KUKA KRL program: nplacestr16RS2.src, nplacestr16RS2.dat

--- nplacestr16RS2.src ---
&ACCESS RVP
&REL 1
&PARAM TEMPLATE = C:\KRC\Roboter\Template\ExpertVorgabe
&PARAM EDITMASK = *
DEF nplacestr16RS2( )
;FOLD INI
  ;FOLD BASISTECH INI
    GLOBAL INTERRUPT DECL 3 WHEN $STOPMESS==TRUE DO IR_STOPM ( )
    INTERRUPT ON 3
    BAS (#INITMOV,0 )
  ;ENDFOLD (BASISTECH INI)
  ;FOLD USER INI
    ;Make your modifications here

  ;ENDFOLD (USER INI)
;ENDFOLD (INI)




SWITCH NumCuring

;*******************************************************
CASE 91601
;*******************************************************
;*** Utilizar para hacer touchup en ptp a continuacion ***;
; 1  Ejecutar Axis_Rob_Move
; 2  Hacer TouchUp en ptp
; 3  Eliminar Axis_Rob_Move y comentarios

Axis_Rob_Move(1.69,-82.8,66.93,14.32,12.14,193,70,50)

;FOLD PTP pWB91601RS2 Vel=100 % PDAT_MESA Tool[10]:AMF1_G1000 Base[7]:BWB4S2;%{PE}%R 5.5.32,%MKUKATPBASIS,%CMOVE,%VPTP,%P 1:PTP, 2:pWB91601RS2, 3:, 5:100, 7:PDAT_MESA
$BWDSTART=FALSE
PDAT_ACT=PPDAT_MESA
FDAT_ACT=FpWB91601RS2
BAS(#PTP_PARAMS,100)
PTP XpWB91601RS2
;ENDFOLD
;*********************************************************;

;***Axis_Rob_Move de ayuda para aproximarse a dejada ***;
; Borrar tras touchup en LIN de dejada
Axis_Rob_Move(-90.22,-57.13,49.23,-5.44,97.37,193.9,20,50)
;*******************************************************;

PTP_OFFS(XP91601RS2, FP91601RS2, 0, -450, 30, 0, 0, 0, #TOOL, 20, 50, 0.0)

Cicle_Grp_M1000 (Inic_Pla_Right)

;***borrar***;
cyltopos(prg_200)
halt
;************;

LIN_OFFS(XP91601RS2, FP91601RS2, 0, 0, 30, 0, 0, 0, #TOOL, 0.1, 50, 0.0)
LIN_OFFS(XP91601RS2, FP91601RS2, 0, 0, 15, 0, 0, 0, #TOOL, 0.1, 50, 0.0)

Cntr_Grp_M1000 (C05C06,RH)

;FOLD LIN P91601RS2 Vel=0.1 m/s LV020Z0 Tool[10]:AMF1_G1000 Base[7]:BWB4S2;%{PE}%R 5.5.32,%MKUKATPBASIS,%CMOVE,%VLIN,%P 1:LIN, 2:P91601RS2, 3:, 5:0.1, 7:V020Z0
$BWDSTART=FALSE
LDAT_ACT=LV020Z0
FDAT_ACT=FP91601RS2
BAS(#CP_PARAMS,0.1)
LIN XP91601RS2
;ENDFOLD

Cntr_Grp_M1000 (AMF09,RLS)
Cyltopos (PRG_51)
Cntr_Grp_M1000 (C07C08,RH)
Cyltopos (PRG_61)
Cntr_Grp_M1000 (AMF10,RLS)
Cntr_Grp_M1000 (C05C06,FREE)
Cntr_Grp_M1000 (C07C08,FREE)
Cyltopos(PRG_88)
LIN_REL{Z -20}#TOOL
Cyltopos (PRG_105)
LIN_REL{Z -30}#TOOL
Cyltopos (PRG_200)

;*** MOVIMIENTOS DE OFFSETS ***;

LIN_OFFS(XP91601RS2, FP91601RS2, 0, 0, -50, 0, 0, 0, #TOOL, 0.3, 50, 0.0)
LIN_OFFS(XP91601RS2, FP91601RS2, 0, -450, -50, 0, 0, 0, #TOOL, 0.3, 50, 0.0)


;******* MEDICION LASER *******;

LIN_OFFS(XPLAS91601RS2_1, FPLAS91601RS2_1, 0, -200, 0, 0, 0, 0, #TOOL, 0.3, 50, 0.0)

cyltopos (prg_61)

;FOLD LIN PLAS91601RS2_1 Vel=0.3 m/s LV020Z0 Tool[10]:AMF1_G1000 Base[7]:BWB4S2;%{PE}%R 5.5.32,%MKUKATPBASIS,%CMOVE,%VLIN,%P 1:LIN, 2:PLAS91601RS2_1, 3:, 5:0.3, 7:V020Z0
$BWDSTART=FALSE
LDAT_ACT=LV020Z0
FDAT_ACT=FPLAS91601RS2_1
BAS(#CP_PARAMS,0.3)
LIN XPLAS91601RS2_1
;ENDFOLD

;Movimimiento de busqueda con laser
;Search( , )

;FOLD LIN PLAS91601RS2_2 Vel=0.3 m/s LV020Z0 Tool[10]:AMF1_G1000 Base[7]:BWB4S2;%{PE}%R 5.5.32,%MKUKATPBASIS,%CMOVE,%VLIN,%P 1:LIN, 2:PLAS91601RS2_2, 3:, 5:0.3, 7:V020Z0
$BWDSTART=FALSE
LDAT_ACT=LV020Z0
FDAT_ACT=FPLAS91601RS2_2
BAS(#CP_PARAMS,0.3)
LIN XPLAS91601RS2_2
;ENDFOLD


;Movimimiento de busqueda con laser
;Search( , )

LIN_OFFS(XPLAS91601RS2_1, FPLAS91601RS2_1, 0, -200, 0, 0, 0, 0, #TOOL, 0.3, 50, 0.0)

;******************************;

;FOLD PTP pWB91601RS2 Vel=100 % PDAT_MESA Tool[10]:AMF1_G1000 Base[7]:BWB4S2;%{PE}%R 5.5.32,%MKUKATPBASIS,%CMOVE,%VPTP,%P 1:PTP, 2:pWB91601RS2, 3:, 5:100, 7:PDAT_MESA
$BWDSTART=FALSE
PDAT_ACT=PPDAT_MESA
FDAT_ACT=FpWB91601RS2
BAS(#PTP_PARAMS,100)
PTP XpWB91601RS2
;ENDFOLD

;*******************************************************
CASE 91603
;*******************************************************
;*** Utilizar para hacer touchup en ptp a continuacion ***;
; 1  Ejecutar Axis_Rob_Move
; 2  Hacer TouchUp en ptp
; 3  Eliminar Axis_Rob_Move y comentarios

Axis_Rob_Move(1.69,-82.8,66.93,14.32,12.14,193,70,50)

;FOLD PTP pWB91603RS2 Vel=100 % PDAT_MESA Tool[10]:AMF1_G1000 Base[7]:BWB4S2;%{PE}%R 5.5.32,%MKUKATPBASIS,%CMOVE,%VPTP,%P 1:PTP, 2:pWB91603RS2, 3:, 5:100, 7:PDAT_MESA
$BWDSTART=FALSE
PDAT_ACT=PPDAT_MESA
FDAT_ACT=FpWB91603RS2
BAS(#PTP_PARAMS,100)
PTP XpWB91603RS2
;ENDFOLD
;*********************************************************;

;***Axis_Rob_Move de ayuda para aproximarse a dejada ***;
; Borrar tras touchup en LIN de dejada
Axis_Rob_Move(-90.22,-57.13,49.23,-5.44,97.37,193.9,20,50)
;*******************************************************;

PTP_OFFS(XP91603RS2, FP91603RS2, 0, -450, 30, 0, 0, 0, #TOOL, 20, 50, 0.0)

Cicle_Grp_M1000 (Inic_Pla_Right)

;***borrar***;
cyltopos(prg_200)
halt
;************;

LIN_OFFS(XP91603RS2, FP91603RS2, 0, 0, 30, 0, 0, 0, #TOOL, 0.1, 50, 0.0)
LIN_OFFS(XP91603RS2, FP91603RS2, 0, 0, 15, 0, 0, 0, #TOOL, 0.1, 50, 0.0)

Cntr_Grp_M1000 (C05C06,RH)

;FOLD LIN P91603RS2 Vel=0.1 m/s LV020Z0 Tool[10]:AMF1_G1000 Base[7]:BWB4S2;%{PE}%R 5.5.32,%MKUKATPBASIS,%CMOVE,%VLIN,%P 1:LIN, 2:P91603RS2, 3:, 5:0.1, 7:V020Z0
$BWDSTART=FALSE
LDAT_ACT=LV020Z0
FDAT_ACT=FP91603RS2
BAS(#CP_PARAMS,0.1)
LIN XP91603RS2
;ENDFOLD

Cntr_Grp_M1000 (AMF09,RLS)
Cyltopos (PRG_51)
Cntr_Grp_M1000 (C07C08,RH)
Cyltopos (PRG_61)
Cntr_Grp_M1000 (AMF10,RLS)
Cntr_Grp_M1000 (C05C06,FREE)
Cntr_Grp_M1000 (C07C08,FREE)
Cyltopos(PRG_88)
LIN_REL{Z -20}#TOOL
Cyltopos (PRG_105)
LIN_REL{Z -30}#TOOL
Cyltopos (PRG_200)

;*** MOVIMIENTOS DE OFFSETS ***;

LIN_OFFS(XP91603RS2, FP91603RS2, 0, 0, -50, 0, 0, 0, #TOOL, 0.3, 50, 0.0)
LIN_OFFS(XP91603RS2, FP91603RS2, 0, -450, -50, 0, 0, 0, #TOOL, 0.3, 50, 0.0)


;******* MEDICION LASER *******;

LIN_OFFS(XPLAS91603RS2_1, FPLAS91603RS2_1, 0, -200, 0, 0, 0, 0, #TOOL, 0.3, 50, 0.0)

cyltopos (prg_61)

;FOLD LIN PLAS91603RS2_1 Vel=0.3 m/s LV020Z0 Tool[10]:AMF1_G1000 Base[7]:BWB4S2;%{PE}%R 5.5.32,%MKUKATPBASIS,%CMOVE,%VLIN,%P 1:LIN, 2:PLAS91603RS2_1, 3:, 5:0.3, 7:V020Z0
$BWDSTART=FALSE
LDAT_ACT=LV020Z0
FDAT_ACT=FPLAS91603RS2_1
BAS(#CP_PARAMS,0.3)
LIN XPLAS91603RS2_1
;ENDFOLD

;Movimimiento de busqueda con laser
;Search( , )

;FOLD LIN PLAS91603RS2_2 Vel=0.3 m/s LV020Z0 Tool[10]:AMF1_G1000 Base[7]:BWB4S2;%{PE}%R 5.5.32,%MKUKATPBASIS,%CMOVE,%VLIN,%P 1:LIN, 2:PLAS91603RS2_2, 3:, 5:0.3, 7:V020Z0
$BWDSTART=FALSE
LDAT_ACT=LV020Z0
FDAT_ACT=FPLAS91603RS2_2
BAS(#CP_PARAMS,0.3)
LIN XPLAS91603RS2_2
;ENDFOLD


;Movimimiento de busqueda con laser
;Search( , )

LIN_OFFS(XPLAS91603RS2_1, FPLAS91603RS2_1, 0, -200, 0, 0, 0, 0, #TOOL, 0.3, 50, 0.0)

;******************************;

;FOLD PTP pWB91603RS2 Vel=100 % PDAT_MESA Tool[10]:AMF1_G1000 Base[7]:BWB4S2;%{PE}%R 5.5.32,%MKUKATPBASIS,%CMOVE,%VPTP,%P 1:PTP, 2:pWB91603RS2, 3:, 5:100, 7:PDAT_MESA
$BWDSTART=FALSE
PDAT_ACT=PPDAT_MESA
FDAT_ACT=FpWB91603RS2
BAS(#PTP_PARAMS,100)
PTP XpWB91603RS2
;ENDFOLD

;*******************************************************
CASE 91605
;*******************************************************
;*** Utilizar para hacer touchup en ptp a continuacion ***;
; 1  Ejecutar Axis_Rob_Move
; 2  Hacer TouchUp en ptp
; 3  Eliminar Axis_Rob_Move y comentarios

Axis_Rob_Move(1.69,-82.8,66.93,14.32,12.14,193,70,50)

;FOLD PTP pWB91605RS2 Vel=100 % PDAT_MESA Tool[10]:AMF1_G1000 Base[7]:BWB4S2;%{PE}%R 5.5.32,%MKUKATPBASIS,%CMOVE,%VPTP,%P 1:PTP, 2:pWB91605RS2, 3:, 5:100, 7:PDAT_MESA
$BWDSTART=FALSE
PDAT_ACT=PPDAT_MESA
FDAT_ACT=FpWB91605RS2
BAS(#PTP_PARAMS,100)
PTP XpWB91605RS2
;ENDFOLD
;*********************************************************;

;***Axis_Rob_Move de ayuda para aproximarse a dejada ***;
; Borrar tras touchup en LIN de dejada
Axis_Rob_Move(-90.22,-57.13,49.23,-5.44,97.37,193.9,20,50)
;*******************************************************;

PTP_OFFS(XP91605RS2, FP91605RS2, 0, -450, 30, 0, 0, 0, #TOOL, 20, 50, 0.0)

Cicle_Grp_M1000 (Inic_Pla_Right)

;***borrar***;
cyltopos(prg_200)
halt
;************;

LIN_OFFS(XP91605RS2, FP91605RS2, 0, 0, 30, 0, 0, 0, #TOOL, 0.1, 50, 0.0)
LIN_OFFS(XP91605RS2, FP91605RS2, 0, 0, 15, 0, 0, 0, #TOOL, 0.1, 50, 0.0)

Cntr_Grp_M1000 (C05C06,RH)

;FOLD LIN P91605RS2 Vel=0.1 m/s LV020Z0 Tool[10]:AMF1_G1000 Base[7]:BWB4S2;%{PE}%R 5.5.32,%MKUKATPBASIS,%CMOVE,%VLIN,%P 1:LIN, 2:P91605RS2, 3:, 5:0.1, 7:V020Z0
$BWDSTART=FALSE
LDAT_ACT=LV020Z0
FDAT_ACT=FP91605RS2
BAS(#CP_PARAMS,0.1)
LIN XP91605RS2
;ENDFOLD

Cntr_Grp_M1000 (AMF09,RLS)
Cyltopos (PRG_51)
Cntr_Grp_M1000 (C07C08,RH)
Cyltopos (PRG_61)
Cntr_Grp_M1000 (AMF10,RLS)
Cntr_Grp_M1000 (C05C06,FREE)
Cntr_Grp_M1000 (C07C08,FREE)
Cyltopos(PRG_88)
LIN_REL{Z -20}#TOOL
Cyltopos (PRG_105)
LIN_REL{Z -30}#TOOL
Cyltopos (PRG_200)

;*** MOVIMIENTOS DE OFFSETS ***;

LIN_OFFS(XP91605RS2, FP91605RS2, 0, 0, -50, 0, 0, 0, #TOOL, 0.3, 50, 0.0)
LIN_OFFS(XP91605RS2, FP91605RS2, 0, -450, -50, 0, 0, 0, #TOOL, 0.3, 50, 0.0)


;******* MEDICION LASER *******;

LIN_OFFS(XPLAS91605RS2_1, FPLAS91605RS2_1, 0, -200, 0, 0, 0, 0, #TOOL, 0.3, 50, 0.0)

cyltopos (prg_61)

;FOLD LIN PLAS91605RS2_1 Vel=0.3 m/s LV020Z0 Tool[10]:AMF1_G1000 Base[7]:BWB4S2;%{PE}%R 5.5.32,%MKUKATPBASIS,%CMOVE,%VLIN,%P 1:LIN, 2:PLAS91605RS2_1, 3:, 5:0.3, 7:V020Z0
$BWDSTART=FALSE
LDAT_ACT=LV020Z0
FDAT_ACT=FPLAS91605RS2_1
BAS(#CP_PARAMS,0.3)
LIN XPLAS91605RS2_1
;ENDFOLD

;Movimimiento de busqueda con laser
;Search( , )

;FOLD LIN PLAS91605RS2_2 Vel=0.3 m/s LV020Z0 Tool[10]:AMF1_G1000 Base[7]:BWB4S2;%{PE}%R 5.5.32,%MKUKATPBASIS,%CMOVE,%VLIN,%P 1:LIN, 2:PLAS91605RS2_2, 3:, 5:0.3, 7:V020Z0
$BWDSTART=FALSE
LDAT_ACT=LV020Z0
FDAT_ACT=FPLAS91605RS2_2
BAS(#CP_PARAMS,0.3)
LIN XPLAS91605RS2_2
;ENDFOLD


;Movimimiento de busqueda con laser
;Search( , )

LIN_OFFS(XPLAS91605RS2_1, FPLAS91605RS2_1, 0, -200, 0, 0, 0, 0, #TOOL, 0.3, 50, 0.0)

;******************************;

;FOLD PTP pWB91605RS2 Vel=100 % PDAT_MESA Tool[10]:AMF1_G1000 Base[7]:BWB4S2;%{PE}%R 5.5.32,%MKUKATPBASIS,%CMOVE,%VPTP,%P 1:PTP, 2:pWB91605RS2, 3:, 5:100, 7:PDAT_MESA
$BWDSTART=FALSE
PDAT_ACT=PPDAT_MESA
FDAT_ACT=FpWB91605RS2
BAS(#PTP_PARAMS,100)
PTP XpWB91605RS2
;ENDFOLD

;*******************************************************
CASE 91607
;*******************************************************
;*** Utilizar para hacer touchup en ptp a continuacion ***;
; 1  Ejecutar Axis_Rob_Move
; 2  Hacer TouchUp en ptp
; 3  Eliminar Axis_Rob_Move y comentarios

Axis_Rob_Move(1.69,-82.8,66.93,14.32,12.14,193,70,50)

;FOLD PTP pWB91607RS2 Vel=100 % PDAT_MESA Tool[10]:AMF1_G1000 Base[7]:BWB4S2;%{PE}%R 5.5.32,%MKUKATPBASIS,%CMOVE,%VPTP,%P 1:PTP, 2:pWB91607RS2, 3:, 5:100, 7:PDAT_MESA
$BWDSTART=FALSE
PDAT_ACT=PPDAT_MESA
FDAT_ACT=FpWB91607RS2
BAS(#PTP_PARAMS,100)
PTP XpWB91607RS2
;ENDFOLD
;*********************************************************;

;***Axis_Rob_Move de ayuda para aproximarse a dejada ***;
; Borrar tras touchup en LIN de dejada
Axis_Rob_Move(-90.22,-57.13,49.23,-5.44,97.37,193.9,20,50)
;*******************************************************;

PTP_OFFS(XP91607RS2, FP91607RS2, 0, -450, 30, 0, 0, 0, #TOOL, 20, 50, 0.0)

Cicle_Grp_M1000 (Inic_Pla_Right)

;***borrar***;
cyltopos(prg_200)
halt
;************;

LIN_OFFS(XP91607RS2, FP91607RS2, 0, 0, 30, 0, 0, 0, #TOOL, 0.1, 50, 0.0)
LIN_OFFS(XP91607RS2, FP91607RS2, 0, 0, 15, 0, 0, 0, #TOOL, 0.1, 50, 0.0)

Cntr_Grp_M1000 (C05C06,RH)

;FOLD LIN P91607RS2 Vel=0.1 m/s LV020Z0 Tool[10]:AMF1_G1000 Base[7]:BWB4S2;%{PE}%R 5.5.32,%MKUKATPBASIS,%CMOVE,%VLIN,%P 1:LIN, 2:P91607RS2, 3:, 5:0.1, 7:V020Z0
$BWDSTART=FALSE
LDAT_ACT=LV020Z0
FDAT_ACT=FP91607RS2
BAS(#CP_PARAMS,0.1)
LIN XP91607RS2
;ENDFOLD

Cntr_Grp_M1000 (AMF09,RLS)
Cyltopos (PRG_51)
Cntr_Grp_M1000 (C07C08,RH)
Cyltopos (PRG_61)
Cntr_Grp_M1000 (AMF10,RLS)
Cntr_Grp_M1000 (C05C06,FREE)
Cntr_Grp_M1000 (C07C08,FREE)
Cyltopos(PRG_88)
LIN_REL{Z -20}#TOOL
Cyltopos (PRG_105)
LIN_REL{Z -30}#TOOL
Cyltopos (PRG_200)

;*** MOVIMIENTOS DE OFFSETS ***;

LIN_OFFS(XP91607RS2, FP91607RS2, 0, 0, -50, 0, 0, 0, #TOOL, 0.3, 50, 0.0)
LIN_OFFS(XP91607RS2, FP91607RS2, 0, -450, -50, 0, 0, 0, #TOOL, 0.3, 50, 0.0)


;******* MEDICION LASER *******;

LIN_OFFS(XPLAS91607RS2_1, FPLAS91607RS2_1, 0, -200, 0, 0, 0, 0, #TOOL, 0.3, 50, 0.0)

cyltopos (prg_61)

;FOLD LIN PLAS91607RS2_1 Vel=0.3 m/s LV020Z0 Tool[10]:AMF1_G1000 Base[7]:BWB4S2;%{PE}%R 5.5.32,%MKUKATPBASIS,%CMOVE,%VLIN,%P 1:LIN, 2:PLAS91607RS2_1, 3:, 5:0.3, 7:V020Z0
$BWDSTART=FALSE
LDAT_ACT=LV020Z0
FDAT_ACT=FPLAS91607RS2_1
BAS(#CP_PARAMS,0.3)
LIN XPLAS91607RS2_1
;ENDFOLD

;Movimimiento de busqueda con laser
;Search( , )

;FOLD LIN PLAS91607RS2_2 Vel=0.3 m/s LV020Z0 Tool[10]:AMF1_G1000 Base[7]:BWB4S2;%{PE}%R 5.5.32,%MKUKATPBASIS,%CMOVE,%VLIN,%P 1:LIN, 2:PLAS91607RS2_2, 3:, 5:0.3, 7:V020Z0
$BWDSTART=FALSE
LDAT_ACT=LV020Z0
FDAT_ACT=FPLAS91607RS2_2
BAS(#CP_PARAMS,0.3)
LIN XPLAS91607RS2_2
;ENDFOLD


;Movimimiento de busqueda con laser
;Search( , )

LIN_OFFS(XPLAS91607RS2_1, FPLAS91607RS2_1, 0, -200, 0, 0, 0, 0, #TOOL, 0.3, 50, 0.0)

;******************************;

;FOLD PTP pWB91607RS2 Vel=100 % PDAT_MESA Tool[10]:AMF1_G1000 Base[7]:BWB4S2;%{PE}%R 5.5.32,%MKUKATPBASIS,%CMOVE,%VPTP,%P 1:PTP, 2:pWB91607RS2, 3:, 5:100, 7:PDAT_MESA
$BWDSTART=FALSE
PDAT_ACT=PPDAT_MESA
FDAT_ACT=FpWB91607RS2
BAS(#PTP_PARAMS,100)
PTP XpWB91607RS2
;ENDFOLD

ENDSWITCH
END

--- nplacestr16RS2.dat ---
DEFDAT nplacestr16RS2
;FOLD EXTERNAL DECLARATIONS;%{PE}%MKUKATPBASIS,%CEXT,%VCOMMON,%P
;FOLD BASISTECH EXT;%{PE}%MKUKATPBASIS,%CEXT,%VEXT,%P
EXT  BAS (BAS_COMMAND  :IN,REAL  :IN )
DECL INT SUCCESS
;ENDFOLD (BASISTECH EXT)
;FOLD USER EXT;%{E}%MKUKATPUSER,%CEXT,%VEXT,%P
;Make here your modifications

;ENDFOLD (USER EXT)
;ENDFOLD (EXTERNAL DECLARATIONS)
DECL E6POS XpWB91601RS2={X 0,Y 0,Z 0,A 0,B 0,C 0,S 2,T 10,E1 0.0,E2 0.0,E3 0.0,E4 0.0,E5 0.0,E6 0.0}
DECL FDAT FpWB91601RS2={TOOL_NO 10,BASE_NO 7,IPO_FRAME #BASE,POINT2[] " ",TQ_STATE FALSE}
;
DECL E6POS XP91601RS2={X 0,Y 0,Z 0,A 0,B 0,C 0,S 2,T 10,E1 0.0,E2 0.0,E3 0.0,E4 0.0,E5 0.0,E6 0.0}
DECL FDAT FP91601RS2={TOOL_NO 10,BASE_NO 7,IPO_FRAME #BASE,POINT2[] " ",TQ_STATE FALSE}
;
DECL E6POS XPLAS91601RS2_1={X 0,Y 0,Z 0,A 0,B 0,C 0,S 2,T 10,E1 0.0,E2 0.0,E3 0.0,E4 0.0,E5 0.0,E6 0.0}
DECL FDAT FPLAS91601RS2_1={TOOL_NO 10,BASE_NO 7,IPO_FRAME #BASE,POINT2[] " ",TQ_STATE FALSE}
DECL E6POS XPLAS91601RS2_2={X 0,Y 0,Z 0,A 0,B 0,C 0,S 2,T 10,E1 0.0,E2 0.0,E3 0.0,E4 0.0,E5 0.0,E6 0.0}
DECL FDAT FPLAS91601RS2_2={TOOL_NO 10,BASE_NO 7,IPO_FRAME #BASE,POINT2[] " ",TQ_STATE FALSE}
;
DECL E6POS XpWB91603RS2={X 0,Y 0,Z 0,A 0,B 0,C 0,S 2,T 10,E1 0.0,E2 0.0,E3 0.0,E4 0.0,E5 0.0,E6 0.0}
DECL FDAT FpWB91603RS2={TOOL_NO 10,BASE_NO 7,IPO_FRAME #BASE,POINT2[] " ",TQ_STATE FALSE}
;
DECL E6POS XP91603RS2={X 0,Y 0,Z 0,A 0,B 0,C 0,S 2,T 10,E1 0.0,E2 0.0,E3 0.0,E4 0.0,E5 0.0,E6 0.0}
DECL FDAT FP91603RS2={TOOL_NO 10,BASE_NO 7,IPO_FRAME #BASE,POINT2[] " ",TQ_STATE FALSE}
;
DECL E6POS XPLAS91603RS2_1={X 0,Y 0,Z 0,A 0,B 0,C 0,S 2,T 10,E1 0.0,E2 0.0,E3 0.0,E4 0.0,E5 0.0,E6 0.0}
DECL FDAT FPLAS91603RS2_1={TOOL_NO 10,BASE_NO 7,IPO_FRAME #BASE,POINT2[] " ",TQ_STATE FALSE}
DECL E6POS XPLAS91603RS2_2={X 0,Y 0,Z 0,A 0,B 0,C 0,S 2,T 10,E1 0.0,E2 0.0,E3 0.0,E4 0.0,E5 0.0,E6 0.0}
DECL FDAT FPLAS91603RS2_2={TOOL_NO 10,BASE_NO 7,IPO_FRAME #BASE,POINT2[] " ",TQ_STATE FALSE}
;
DECL E6POS XpWB91605RS2={X 0,Y 0,Z 0,A 0,B 0,C 0,S 2,T 10,E1 0.0,E2 0.0,E3 0.0,E4 0.0,E5 0.0,E6 0.0}
DECL FDAT FpWB91605RS2={TOOL_NO 10,BASE_NO 7,IPO_FRAME #BASE,POINT2[] " ",TQ_STATE FALSE}
;
DECL E6POS XP91605RS2={X 0,Y 0,Z 0,A 0,B 0,C 0,S 2,T 10,E1 0.0,E2 0.0,E3 0.0,E4 0.0,E5 0.0,E6 0.0}
DECL FDAT FP91605RS2={TOOL_NO 10,BASE_NO 7,IPO_FRAME #BASE,POINT2[] " ",TQ_STATE FALSE}
;
DECL E6POS XPLAS91605RS2_1={X 0,Y 0,Z 0,A 0,B 0,C 0,S 2,T 10,E1 0.0,E2 0.0,E3 0.0,E4 0.0,E5 0.0,E6 0.0}
DECL FDAT FPLAS91605RS2_1={TOOL_NO 10,BASE_NO 7,IPO_FRAME #BASE,POINT2[] " ",TQ_STATE FALSE}
DECL E6POS XPLAS91605RS2_2={X 0,Y 0,Z 0,A 0,B 0,C 0,S 2,T 10,E1 0.0,E2 0.0,E3 0.0,E4 0.0,E5 0.0,E6 0.0}
DECL FDAT FPLAS91605RS2_2={TOOL_NO 10,BASE_NO 7,IPO_FRAME #BASE,POINT2[] " ",TQ_STATE FALSE}
;
DECL E6POS XpWB91607RS2={X 0,Y 0,Z 0,A 0,B 0,C 0,S 2,T 10,E1 0.0,E2 0.0,E3 0.0,E4 0.0,E5 0.0,E6 0.0}
DECL FDAT FpWB91607RS2={TOOL_NO 10,BASE_NO 7,IPO_FRAME #BASE,POINT2[] " ",TQ_STATE FALSE}
;
DECL E6POS XP91607RS2={X 0,Y 0,Z 0,A 0,B 0,C 0,S 2,T 10,E1 0.0,E2 0.0,E3 0.0,E4 0.0,E5 0.0,E6 0.0}
DECL FDAT FP91607RS2={TOOL_NO 10,BASE_NO 7,IPO_FRAME #BASE,POINT2[] " ",TQ_STATE FALSE}
;
DECL E6POS XPLAS91607RS2_1={X 0,Y 0,Z 0,A 0,B 0,C 0,S 2,T 10,E1 0.0,E2 0.0,E3 0.0,E4 0.0,E5 0.0,E6 0.0}
DECL FDAT FPLAS91607RS2_1={TOOL_NO 10,BASE_NO 7,IPO_FRAME #BASE,POINT2[] " ",TQ_STATE FALSE}
DECL E6POS XPLAS91607RS2_2={X 0,Y 0,Z 0,A 0,B 0,C 0,S 2,T 10,E1 0.0,E2 0.0,E3 0.0,E4 0.0,E5 0.0,E6 0.0}
DECL FDAT FPLAS91607RS2_2={TOOL_NO 10,BASE_NO 7,IPO_FRAME #BASE,POINT2[] " ",TQ_STATE FALSE}
;
ENDDAT
